PROGRAM MAIN
VAR
	test: BOOL;
	test2: INT;
END_VAR

END_PROGRAM

(* stored: Version 1.1.0.1, ProductVersion 3.1.4020.6
   POU MAIN: Id {ab6847ec-51d6-424e-b5cc-ca01f095b99f}, SpecialFunc None *)
